TYPE TcoDatamanResultsStatus_v_5_x_x : 
STRUCT
    Decoding AT %I* : BOOL;
    DecodeComplete AT %I* : BOOL;
    ResultsBufferOverrun AT %I* : BOOL;
    ResultsAvailable AT %I* : BOOL;
    ErrorDetected AT %I* : BOOL;
END_STRUCT
END_TYPE

(* stored: Version 1.1.0.1, ProductVersion 3.1.4024.11
   DUT TcoDatamanResultsStatus_v_5_x_x: Id {af59c109-c71c-4a20-b5ce-79be06027ed4} *)
